{attribute clr [Container(Layout.Stack)]}
{attribute clr [Group(Layout.Scroll)]}
TYPE CUTechnologicalDataBase EXTENDS TcoCore.TcoStruct :
STRUCT
	
END_STRUCT
END_TYPE

(* stored: Version 1.1.0.1
   DUT CUTechnologicalDataBase: Id {7f1b525b-56fa-09a1-1f2d-f6d3ae7fbaf7} *)
